(*			
	RAFALOS
	Rafał Osajda		19.09.2025		TC 4024.66
	
*)
FUNCTION_BLOCK FB_BaseFlag IMPLEMENTS ITF_BaseFlag
VAR
END_VAR

END_FUNCTION_BLOCK

(* stored: Version 1.1.0.1
   POU FB_BaseFlag: Id {4cccc323-b44e-0e45-096d-9e86741e033e}, SpecialFunc None *)
